FUNCTION_BLOCK Starting EXTENDS Vanguard_WaferDetection.State
VAR
	StartupState : INT;
	ChannelControl : I_VisionChannelControl;
END_VAR

METHOD Executing : BOOL
CASE StartupState OF
// 	0: //Unknown conditions
// 		IF SUCCEEDED(GVL_Vision.LabelProcess.LoadRecipe(WaferDetectRecipe)) THEN
// 			SystemReady := TRUE;
// 			StartupState := 1;
// 		END_IF

	0:
		IF ChannelControl.StartVision() THEN
			StartupState := 1;
		END_IF
	1:
		StartupState := 0;
		Executing := TRUE;
END_CASE
END_METHOD

METHOD SetDependencies : BOOL
VAR_INPUT
	Control : I_VisionChannelControl;
END_VAR
ChannelControl := Control;
END_METHOD

END_FUNCTION_BLOCK

(* stored: Version 1.1.0.1
   POU Starting: Id {a6366843-b758-4595-9d46-48cc57b0118e}, SpecialFunc None
   Method Executing: Id {f346418a-a3d9-4176-a409-28486b55d633}
   Method SetDependencies: Id {eb43ab81-e9c2-4ceb-a702-e9f0d9133a11} *)
